Staubli VAL3: RobotMotion.pgx

program RobotMotion()
  local num nNummove
begin

  movej(pfrmCad[0],tTool,mNomSpeed)
  waitEndMove()
  bSignal=true
  nNummove=0

  do
    movej(pfrmCad[nNummove],tTool,mNomSpeed)
    nNumrecord=nNumrecord+1

    if nNummove==600
      bTxt1=true
    endIf
    if nNummove==1100
      bTxt2=true
    endIf
    if nNummove==100
      bTxt3=true
    endIf
    delay(0)
    if nNummove==1499
      nNummove=0
    else
      nNummove=nNummove+1
    endIf
  until nNumrecord==nNumTotal
  waitEndMove()
  bSignal=false
  taskKill("PositionTrigger")
  ndelay=clock()-ntime

end
